Staubli VAL3: sendAck.pgx

program sendAck(num id)
  local num buffer[3]
begin
  buffer[0] = MAGIC_HEADER
  buffer[1] = 128
  buffer[2] = id
  sioSet(socket, buffer)
end
